TYPE WaferDetectionVisionRecipe :
STRUCT
	MedianFilterSize : UDINT;
END_STRUCT
END_TYPE

(* stored: Version 1.1.0.1
   DUT WaferDetectionVisionRecipe: Id {e8dc570e-fc7e-47f6-b5d7-bfafaece0eb8} *)
